FUNCTION_BLOCK FB_MGMT_Ablaufsteuerung
VAR_IN_OUT
	Zustand				: ST_FB_MGMT_Zustand;
	Stellwert			: ST_FB_MGMT_Stellwert;
	Steuerung			: ST_FB_MGMT_Steuerung;
END_VAR
VAR_INPUT
END_VAR
VAR_OUTPUT
END_VAR
VAR
END_VAR

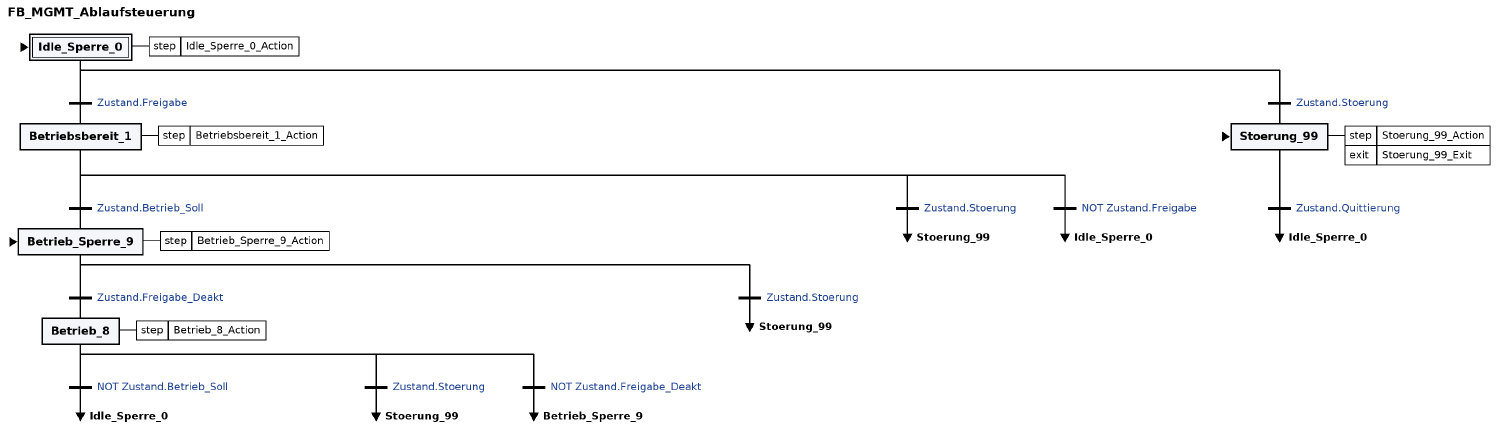
INITIAL_STEP Idle_Sperre_0:
    Idle_Sperre_0_Action(N);  // step action
END_STEP
TRANSITION FROM Idle_Sperre_0 TO Betriebsbereit_1
    := Zustand.Freigabe;
END_TRANSITION
TRANSITION FROM Idle_Sperre_0 TO Stoerung_99
    := Zustand.Stoerung;
END_TRANSITION
STEP Stoerung_99:
    Stoerung_99_Action(N);  // step action
    Stoerung_99_Exit(P0);  // exit action
END_STEP
TRANSITION FROM Stoerung_99 TO Idle_Sperre_0
    := Zustand.Quittierung;
END_TRANSITION
STEP Betriebsbereit_1:
    Betriebsbereit_1_Action(N);  // step action
END_STEP
TRANSITION FROM Betriebsbereit_1 TO Betrieb_Sperre_9
    := Zustand.Betrieb_Soll;
END_TRANSITION
TRANSITION FROM Betriebsbereit_1 TO Stoerung_99
    := Zustand.Stoerung;
END_TRANSITION
TRANSITION FROM Betriebsbereit_1 TO Idle_Sperre_0
    := NOT Zustand.Freigabe;
END_TRANSITION
STEP Betrieb_Sperre_9:
    Betrieb_Sperre_9_Action(N);  // step action
END_STEP
TRANSITION FROM Betrieb_Sperre_9 TO Betrieb_8
    := Zustand.Freigabe_Deakt;
END_TRANSITION
TRANSITION FROM Betrieb_Sperre_9 TO Stoerung_99
    := Zustand.Stoerung;
END_TRANSITION
STEP Betrieb_8:
    Betrieb_8_Action(N);  // step action
END_STEP
TRANSITION FROM Betrieb_8 TO Idle_Sperre_0
    := NOT Zustand.Betrieb_Soll;
END_TRANSITION
TRANSITION FROM Betrieb_8 TO Stoerung_99
    := Zustand.Stoerung;
END_TRANSITION
TRANSITION FROM Betrieb_8 TO Betrieb_Sperre_9
    := NOT Zustand.Freigabe_Deakt;
END_TRANSITION

ACTION Betrieb_8_Action:
(* Stellwert setzen *)
Stellwert.Betrieb				:= TRUE;
Zustand.Betrieb				:= TRUE;

(* Zustand setzen *)
Zustand.Status				:= E_MGMT_Zustand_Status_Betrieb;
END_ACTION

ACTION Betrieb_Sperre_9_Action:
(* Stellwert setzen *)
Stellwert.Betrieb				:= TRUE;
Zustand.Betrieb				:= TRUE;

(* Zustand setzen *)
Zustand.Status				:= E_MGMT_Zustand_Status_Betrieb_Sperre;
END_ACTION

ACTION Betriebsbereit_1_Action:
(* Stellwert setzen *)
Stellwert.Betrieb		:= FALSE;
Zustand.Betrieb		:= FALSE;

(* Zustand setzen *)
Zustand.Status			:= E_MGMT_Zustand_Status_Betriebsbereit;
END_ACTION

ACTION Idle_Sperre_0_Action:
(* Stellwert setzen *)
Stellwert.Betrieb		:= FALSE;
Zustand.Betrieb			:= FALSE;

(* Zustand setzen *)
Zustand.Status				:= E_MGMT_Zustand_Status_Idle_Sperre;

(* Quittierungszustand auf False setzen, damit das System bei einer erneuten Störung nicht direkt wieder angeschaltet wird *)
Steuerung.Quittierung	:= FALSE;
END_ACTION

ACTION Stoerung_99_Action:
(* Stellwert setzen *)
Stellwert.Betrieb			:= FALSE;
Zustand.Betrieb			:= FALSE;

(* Zustand setzen *)
Zustand.Stoerung			:= TRUE;
Zustand.Status			:= E_MGMT_Zustand_Status_Stoerung;
END_ACTION

ACTION Stoerung_99_Exit:
Zustand.Stoerung	:= FALSE;
END_ACTION

END_FUNCTION_BLOCK

(* stored: Version 1.1.0.1, ProductVersion 3.1.4024.9
   POU FB_MGMT_Ablaufsteuerung: Id {59daa17c-eefb-4ce3-868f-29b5ed862c19}, SpecialFunc None
   Action Betrieb_8_Action: Id {3027da9d-c2bc-49d5-9930-d7582964389e}
   Action Betrieb_Sperre_9_Action: Id {11056bd5-e42a-4d27-a22a-d016ef9b8c65}
   Action Betriebsbereit_1_Action: Id {a1cd02c5-f2b1-46cc-b7b8-552b2dd388be}
   Action Idle_Sperre_0_Action: Id {a38c7b35-3e3a-4b3e-9d61-e59d9147eaf7}
   Action Stoerung_99_Action: Id {af82e2d6-09fb-4e4b-be5c-297384f85b93}
   Action Stoerung_99_Exit: Id {da698741-cbe6-4f7d-a689-01172b6945a4} *)
